(*
  FUNCTION_BLOCK FB_LevelControl
  Purpose:
    - Level control with Auto/Manual output (0..100 %).
    - PID (OSCAT CTRL_PID) with bumpless transfer.
    - Optional PT1 input filter.
    - VFD supervision: ready, fault, run feedback with timeout.
    - Safety supervision: E-Stop/guards/safety chain => immediate stop anywhere.
    - Interlocks (process permissives) => NORMAL STOP ONLY.
    - Minimum level supervision with hysteresis & debounce (stop/hold/restart).
    - deviceState: human-readable state string.

  States:
    0=Idle, 10=Starting, 20=Running, 90=Stopping
*)

FUNCTION_BLOCK FB_LevelControl
VAR_INPUT
    // ===== Sequence commands =====
    startCommand            : BOOL;            // Start command
    stopCommand             : BOOL;            // Stop command

    // ===== Mode =====
    autoMode                : BOOL;            // TRUE=Automatic / FALSE=Manual

    // ===== Process signals (LEVEL) =====
    levelFeedbackEng        : REAL;            // Level feedback (engineering units)
    levelSetpointEng        : REAL;            // Setpoint in engineering units

    // ===== Manual output (direct % to final element) =====
    manualOutputPct         : REAL;            // 0..100% manual output

    // ===== PID parameters (OSCAT CTRL_PID) =====
    kp                      : REAL := 1.0;     // proportional gain
    tn                      : REAL := 8.0;     // integral time [s]
    tv                      : REAL := 0.0;     // derivative time [s]

    // ===== Output limits & offset =====
    outLowLimitPct          : REAL := 0.0;
    outHighLimitPct         : REAL := 100.0;
    outputOffsetPct         : REAL := 0.0;     // added to final output

    // ===== PID housekeeping =====
    resetPID                : BOOL;            // reset integrator

    // ===== Input filter (OSCAT PT1) =====
    enableInputFilter       : BOOL := TRUE;
    inputFilterTime         : TIME := T#500ms;
    inputFilterGainK        : REAL := 1.0;

    // ===== Optional scaling (engineering <-> %) =====
    enableScaling           : BOOL := TRUE;
    lvlLoEng                : REAL := 0.0;
    lvlHiEng                : REAL := 100.0;

    // ===== VFD interface & supervision =====
    vfdReady                : BOOL;            // VFD ready/healthy
    vfdRunFeedback          : BOOL;            // VFD RUN feedback
    vfdFaultFeedback        : BOOL;            // VFD fault feedback
    vfdRunFbTimeout         : TIME := T#5s;    // Timeout to receive RUN FB after start

    // ===== SAFETY (true safety only) =====
    safetyOk                : BOOL := TRUE;    // Safety relay / chain OK
    estopOk                 : BOOL := TRUE;    // E-Stop loop OK
    guardClosedOk           : BOOL := TRUE;    // Doors/guards closed

    // ===== INTERLOCKS (process permissives) — NORMAL STOP ONLY =====
    interlock1              : BOOL := TRUE;
    interlock2              : BOOL := TRUE;
    interlock3              : BOOL := TRUE;
    interlock4              : BOOL := TRUE;
    interlock5              : BOOL := TRUE;
    interlock6              : BOOL := TRUE;

    // ===== Minimum level supervision (process permissive) =====
    minLevelEnable          : BOOL := TRUE;    // Enable low-level stop/hold logic
    minLevelStopEng         : REAL := 10.0;    // Trip threshold (Eng units) => stop & hold
    minLevelRestartEng      : REAL := 12.0;    // Release threshold (Eng units) => auto restart
    minLevelTripTime        : TIME := T#1s;    // Level < StopEng for this long to trip
    minLevelReleaseTime     : TIME := T#1s;    // Level > RestartEng for this long to release
END_VAR

VAR_OUTPUT
    running                 : BOOL;            // TRUE only in RUN (use to release other devices)
    controlOutputPct        : REAL;            // 0..100 %
    pidDiff                 : REAL;            // SET - ACT (post-scaling)
    pidLimited              : BOOL;            // TRUE if saturated
    deviceState             : STRING(80);      // Human-readable state
    vfdStartCmdOut          : BOOL;            // Asserted in Starting/Running (VFD START)
    minLevelHoldActive      : BOOL;            // TRUE while in low-level hold
END_VAR

VAR
    // State
    step                    : INT;             // 0=Idle,10=Starting,20=Running,90=Stopping
    startOld                : BOOL;
    rStart                  : BOOL;

    // Internals
    manualCmd               : REAL;
    yPID                    : REAL;

    // Filtered PV (engineering)
    levelFeedbackEngFilt    : REAL;

    // PV/SP in %
    pvPct                   : REAL;
    spPct                   : REAL;

    // Timers / supervision
    tonRunFbWait            : TON;

    // Minimum level timers/flags
    minLevelBelow           : BOOL;
    minLevelAboveRestart    : BOOL;
    tonMinLevelTrip         : TON;
    tonMinLevelRelease      : TON;

    // Instances
    instPID                 : CTRL_PID;
    instPT1                 : FT_PT1;

    // Safety aggregation
    allSafetyOK             : BOOL;

    // Interlock aggregation (process-only)
    anyInterlockOpen        : BOOL;
END_VAR



// ============================ Edges ============================
rStart := startCommand AND NOT startOld;
startOld := startCommand;


// ============================ Aggregations =====================
allSafetyOK := safetyOk AND estopOk AND guardClosedOk;
anyInterlockOpen := NOT (interlock1 AND interlock2 AND interlock3 AND interlock4 AND interlock5 AND interlock6);

// Default each cycle
vfdStartCmdOut := FALSE;


// ============================ Minimum level supervision ============================
// Compare using current engineering PV (raw). If preferred, swap to levelFeedbackEngFilt.
minLevelBelow        := (levelFeedbackEng <  minLevelStopEng);
minLevelAboveRestart := (levelFeedbackEng >  minLevelRestartEng);

IF minLevelEnable THEN
    // Trip debounce
    tonMinLevelTrip(IN := minLevelBelow, PT := minLevelTripTime);
    // Release debounce
    tonMinLevelRelease(IN := minLevelAboveRestart, PT := minLevelReleaseTime);

    // Latch HOLD on trip, clear on release
    IF tonMinLevelTrip.Q THEN
        minLevelHoldActive := TRUE;
    END_IF;
    IF tonMinLevelRelease.Q THEN
        minLevelHoldActive := FALSE;
    END_IF;
ELSE
    tonMinLevelTrip(IN := FALSE);
    tonMinLevelRelease(IN := FALSE);
    minLevelHoldActive := FALSE;
END_IF;


// ============================ Immediate stop / safety/fault guards ============
IF stopCommand THEN
    controlOutputPct := 0.0;
    running := FALSE;
    deviceState := 'Stopping (Stop command)';
    step := 90;
END_IF;

IF vfdFaultFeedback THEN
    deviceState := 'Fault from VFD';
    step := 90;
END_IF;

IF NOT allSafetyOK THEN
    deviceState := 'Stopping: Safety chain open';
    step := 90;
END_IF;


// ============================ State machine =====================
CASE step OF
    // ------------------------------------------------------------
    0: // Idle
        running := FALSE;
        controlOutputPct := 0.0;
        deviceState := 'Idle';
        vfdStartCmdOut := FALSE;

        // Start request
        IF rStart AND NOT stopCommand THEN
            // Safety must be OK; VFD must be ready; min level must not be holding
            IF NOT allSafetyOK THEN
                deviceState := 'Start blocked: Safety not OK';
                step := 0;
            ELSIF NOT vfdReady THEN
                deviceState := 'Start blocked: VFD not ready';
                step := 0;
            ELSIF minLevelEnable AND minLevelHoldActive THEN
                deviceState := 'Start blocked: Low level hold';
                step := 0;
            ELSE
                deviceState := 'Starting';
                vfdStartCmdOut := TRUE;                   // send START to VFD
                tonRunFbWait(IN := TRUE, PT := vfdRunFbTimeout);
                step := 10;
            END_IF
        END_IF

    // ------------------------------------------------------------
    10: // Starting (await RUN feedback)
        running := FALSE;
        deviceState := 'Starting (await RUN fb)';
        vfdStartCmdOut := TRUE;

        // Safety/fault during start => stop
        IF NOT allSafetyOK THEN
            tonRunFbWait(IN := FALSE);
            deviceState := 'Stopping: Safety chain open';
            vfdStartCmdOut := FALSE;
            step := 90;

        ELSIF vfdFaultFeedback THEN
            tonRunFbWait(IN := FALSE);
            deviceState := 'Fault from VFD';
            vfdStartCmdOut := FALSE;
            step := 90;

        // Interlocks are normal stop only
        ELSIF anyInterlockOpen THEN
            tonRunFbWait(IN := FALSE);
            deviceState := 'Stopping: Interlock open';
            vfdStartCmdOut := FALSE;
            step := 90;

        // Minimum level HOLD => normal stop
        ELSIF minLevelEnable AND minLevelHoldActive THEN
            tonRunFbWait(IN := FALSE);
            deviceState := 'Stopping: Low level hold';
            vfdStartCmdOut := FALSE;
            step := 90;

        // RUN fb arrived
        ELSIF vfdRunFeedback THEN
            tonRunFbWait(IN := FALSE);
            step := 20;

        // Timeout
        ELSIF tonRunFbWait.Q THEN
            tonRunFbWait(IN := FALSE);
            deviceState := 'Start failed: RUN feedback timeout';
            vfdStartCmdOut := FALSE;
            step := 90;
        END_IF

    // ------------------------------------------------------------
    20: // Running (control loop)
        running := TRUE;               // release other devices with this
        deviceState := 'Running';
        vfdStartCmdOut := TRUE;

        // Supervision
        IF NOT allSafetyOK THEN
            deviceState := 'Stopping: Safety chain open';
            vfdStartCmdOut := FALSE;
            step := 90;

        ELSIF vfdFaultFeedback THEN
            deviceState := 'Fault from VFD';
            vfdStartCmdOut := FALSE;
            step := 90;

        ELSIF NOT vfdReady THEN
            deviceState := 'Stopping: VFD not ready';
            vfdStartCmdOut := FALSE;
            step := 90;

        ELSIF NOT vfdRunFeedback THEN
            deviceState := 'Stopping: RUN feedback lost';
            vfdStartCmdOut := FALSE;
            step := 90;

        // INTERLOCKS → NORMAL STOP ONLY
        ELSIF anyInterlockOpen THEN
            deviceState := 'Stopping: Interlock open';
            vfdStartCmdOut := FALSE;
            step := 90;

        // Minimum level HOLD → NORMAL STOP
        ELSIF minLevelEnable AND minLevelHoldActive THEN
            deviceState := 'Stopping: Low level hold';
            vfdStartCmdOut := FALSE;
            step := 90;

        ELSIF stopCommand THEN
            deviceState := 'Stopping (Stop command)';
            vfdStartCmdOut := FALSE;
            step := 90;

        ELSE
            // ---- Input filtering (PT1) ----
            IF enableInputFilter THEN
                instPT1(in := levelFeedbackEng, T := inputFilterTime, K := inputFilterGainK, out => levelFeedbackEngFilt);
            ELSE
                levelFeedbackEngFilt := levelFeedbackEng;
            END_IF

            // ---- Engineering -> % scaling ----
            IF enableScaling THEN
                pvPct := _ScaleToPct(levelFeedbackEngFilt, lvlLoEng, lvlHiEng);
                spPct := _ScaleToPct(levelSetpointEng,     lvlLoEng, lvlHiEng);
            ELSE
                pvPct := levelFeedbackEngFilt;    // already %
                spPct := levelSetpointEng;        // already %
            END_IF

            // ---- Manual path and PID with bumpless transfer ----
            manualCmd := LIMIT(0.0, manualOutputPct, 100.0);

            instPID(
                ACT := pvPct,
                SET := spPct,
                M_I := manualCmd,
                MAN := NOT autoMode,
                RST := resetPID,
                KP  := kp,
                TN  := tn,
                TV  := tv,
                LL  := outLowLimitPct,
                LH  := outHighLimitPct,
                Y   => yPID,
                DIFF=> pidDiff,
                LIM => pidLimited
            );

            // Mode select, offset, clamp
            IF autoMode THEN
                controlOutputPct := yPID;
            ELSE
                controlOutputPct := manualCmd;
            END_IF
            controlOutputPct := LIMIT(outLowLimitPct, controlOutputPct + outputOffsetPct, outHighLimitPct);
        END_IF

    // ------------------------------------------------------------
    90: // Stopping (normal, de-energize)
        running := FALSE;
        controlOutputPct := 0.0;
        vfdStartCmdOut := FALSE;
        tonRunFbWait(IN := FALSE);

        // Return to Idle once stop released and safety OK
        IF NOT stopCommand AND allSafetyOK THEN
            deviceState := 'Idle';
            step := 0;
        END_IF

    // ------------------------------------------------------------
    ELSE
        running := FALSE;
        controlOutputPct := 0.0;
        deviceState := 'Idle';
        vfdStartCmdOut := FALSE;
        step := 0;
END_CASE

// ============================ Helper ============================
METHOD PRIVATE _ScaleToPct : REAL
VAR_INPUT
    xEng  : REAL;  // value in engineering units
    loEng : REAL;  // min eng
    hiEng : REAL;  // max eng
END_VAR
VAR
    span : REAL;
    pct  : REAL;
END_VAR

span := hiEng - loEng;
IF span = 0.0 THEN
    _ScaleToPct := 0.0; // avoid div by zero
ELSE
    pct := (xEng - loEng) / span * 100.0;
    _ScaleToPct := LIMIT(0.0, pct, 100.0);
END_IF
END_METHOD

END_FUNCTION_BLOCK

(* stored: Version 1.1.0.1, ProductVersion 3.1.4024.15
   POU FB_LevelControl: Id {a29e515f-6d43-40bf-8407-f8944f7ce5b0}, SpecialFunc None
   Method _ScaleToPct: Id {e4e5c673-50b3-4c49-aecf-5f846c890a68} *)
